(* Logix 5000 project; controller cal1632 1756-L62 rev 16.20; software revision 16.05; part 38 of 57 *)
(* tags used below, declared in another part *)
   FAULT : BOOL;
   p01_param_oven_timer_presets : DINT[32];
   p01_recipe_active : recipe;
   p01r09 : routine;
   p01r09_pb_global_reset : BOOL;
   p02_dint_from_hmi : hmi_dint;
   p02_real_from_hmi : hmi_real;
   p23_ao_servo_ds_jog_vel_cmd : REAL;
   p23_ao_servo_ds_position_cmd : REAL;
   p23_ao_servo_ds_velocity_cmd : REAL;
   p23_ao_servo_ds_zero_offset : REAL;
   p23_ao_servo_os_jog_vel_cmd : REAL;
   p23_ao_servo_os_position_cmd : REAL;
   p23_ao_servo_os_velocity_cmd : REAL;
   p23_ao_servo_os_zero_offset : REAL;
   p23_di_servo_ds : servo_di;
   p23_di_servo_os : servo_di;
   p23_di_vfd_jog_fwd : BOOL;
   p23_di_vfd_jog_rev : BOOL;
   p23_do_servo_ds : servo_do;
   p23_do_servo_os : servo_do;
   p23_param_lfl_hhl : REAL;
   p23_param_lfl_hl : REAL;
   p23_param_zone_pressure : REAL;
   p23r09 : routine;
   p23r09_mode_run : BOOL;
   p23r09_timer_fault : TIMER[4];
   p23r09_web_wet_ctrl_toggle : SYS_Toggle;
   p23r10 : routine;
   p23r10_timer_fault : TIMER[4];
   p23r10_timer_warning : TIMER[4];
   p23r11 : routine;
   p23r11_impreg_gap_os : REAL;
   p23r11_offsets : REAL[100];
   p23r11_permissive_jog : BOOL;
   p23r11_pos_offset : REAL;
   p23r11_request_jog_fwd : BOOL;
   p23r11_request_jog_rev : BOOL;
   p23r11_request_position : BOOL;
   p23r11_request_start : BOOL;
   p23r11_request_zero : BOOL;
   p23r11_selected_position : REAL;
   p23r11_servo_not_ready : BOOL;
   p23r11_servo_status_ab : BOOL;
   p23r11_servo_status_af : BOOL;
   p23r11_servo_status_bb : BOOL;
   p23r11_timer : TIMER[4];
   p23r11_timer_fault : TIMER[4];
   p23r11_timer_warning : TIMER[4];
   p23r12 : routine;
   p23r12_impreg_gap_ds : REAL;
   p23r12_offsets : REAL[100];
   p23r12_permissive_jog : BOOL;
   p23r12_pos_offset : REAL;
   p23r12_request_jog_fwd : BOOL;
   p23r12_request_jog_rev : BOOL;
   p23r12_request_position : BOOL;
   p23r12_request_start : BOOL;
   p23r12_request_zero : BOOL;
   p23r12_selected_position : REAL;
   p23r12_servo_not_ready : BOOL;
   p23r12_servo_status_ab : BOOL;
   p23r12_servo_status_af : BOOL;
   p23r12_servo_status_bb : BOOL;
   p23r12_timer : TIMER[4];
   p23r12_timer_fault : TIMER[4];
   p23r12_timer_warning : TIMER[4];
   p23r15_pid_tension_control : BOOL;
(* P23_Impreg, continued *)

ROUTINE R09_Modes   (* ladder *)
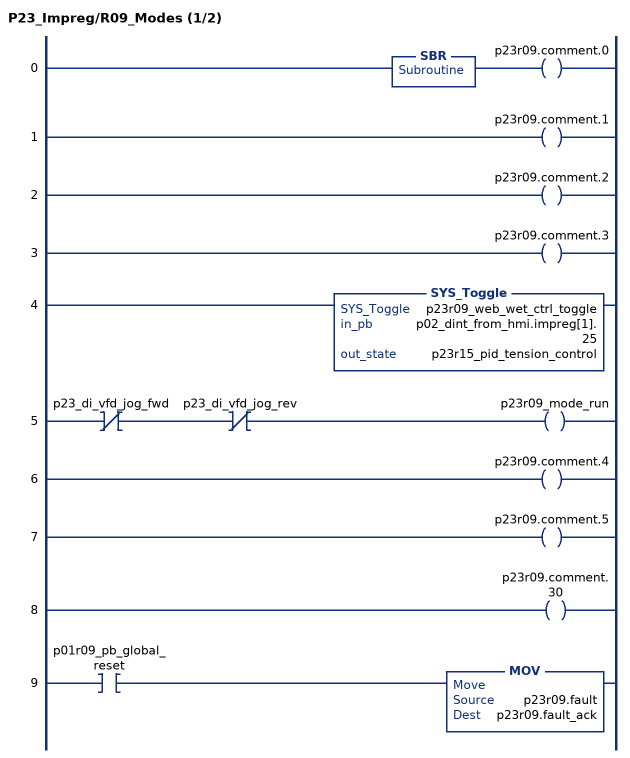
   0: SBR()OTE(p23r09.comment.0);
   1: OTE(p23r09.comment.1);
   2: OTE(p23r09.comment.2);
   3: OTE(p23r09.comment.3);
   4: SYS_Toggle(p23r09_web_wet_ctrl_toggle,p02_dint_from_hmi.impreg[1].25,p23r15_pid_tension_control);
   5: XIO(p23_di_vfd_jog_fwd)XIO(p23_di_vfd_jog_rev)OTE(p23r09_mode_run);
   6: OTE(p23r09.comment.4);
   7: OTE(p23r09.comment.5);
   8: OTE(p23r09.comment.30);
   9: XIC(p01r09_pb_global_reset)MOV(p23r09.fault,p23r09.fault_ack);
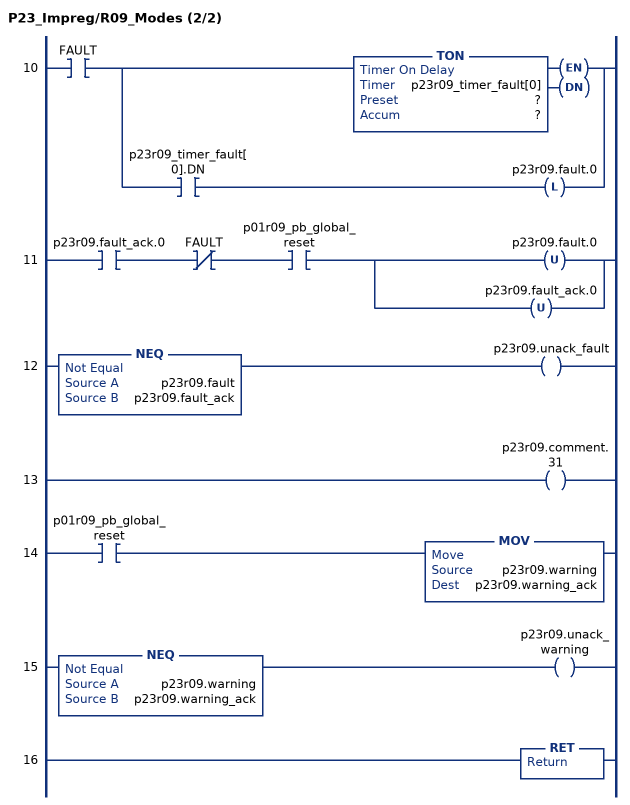
   10: XIC(FAULT)[TON(p23r09_timer_fault[0],?,?) ,XIC(p23r09_timer_fault[0].DN) OTL(p23r09.fault.0) ];
   11: XIC(p23r09.fault_ack.0)XIO(FAULT)XIC(p01r09_pb_global_reset)[OTU(p23r09.fault.0) ,OTU(p23r09.fault_ack.0) ];
   12: NEQ(p23r09.fault,p23r09.fault_ack)OTE(p23r09.unack_fault);
   13: OTE(p23r09.comment.31);
   14: XIC(p01r09_pb_global_reset)MOV(p23r09.warning,p23r09.warning_ack);
   15: NEQ(p23r09.warning,p23r09.warning_ack)OTE(p23r09.unack_warning);
   16: RET();
END_ROUTINE

ROUTINE R10_Parameters   (* ladder *)
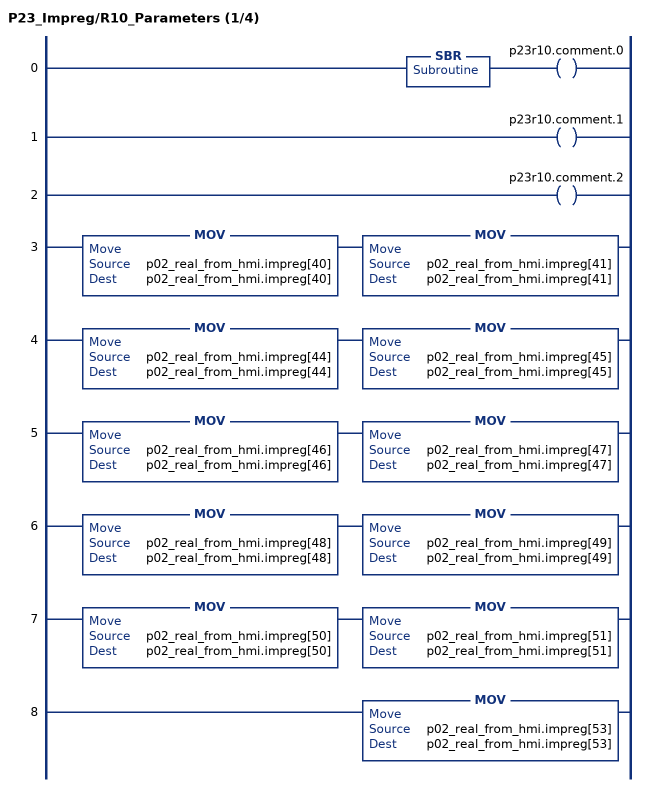
   0: SBR()OTE(p23r10.comment.0);
   1: OTE(p23r10.comment.1);
   2: OTE(p23r10.comment.2);
   3: MOV(p02_real_from_hmi.impreg[40],p02_real_from_hmi.impreg[40])MOV(p02_real_from_hmi.impreg[41],p02_real_from_hmi.impreg[41]);
   4: MOV(p02_real_from_hmi.impreg[44],p02_real_from_hmi.impreg[44])MOV(p02_real_from_hmi.impreg[45],p02_real_from_hmi.impreg[45]);
   5: MOV(p02_real_from_hmi.impreg[46],p02_real_from_hmi.impreg[46])MOV(p02_real_from_hmi.impreg[47],p02_real_from_hmi.impreg[47]);
   6: MOV(p02_real_from_hmi.impreg[48],p02_real_from_hmi.impreg[48])MOV(p02_real_from_hmi.impreg[49],p02_real_from_hmi.impreg[49]);
   7: MOV(p02_real_from_hmi.impreg[50],p02_real_from_hmi.impreg[50])MOV(p02_real_from_hmi.impreg[51],p02_real_from_hmi.impreg[51]);
   8: MOV(p02_real_from_hmi.impreg[53],p02_real_from_hmi.impreg[53]);
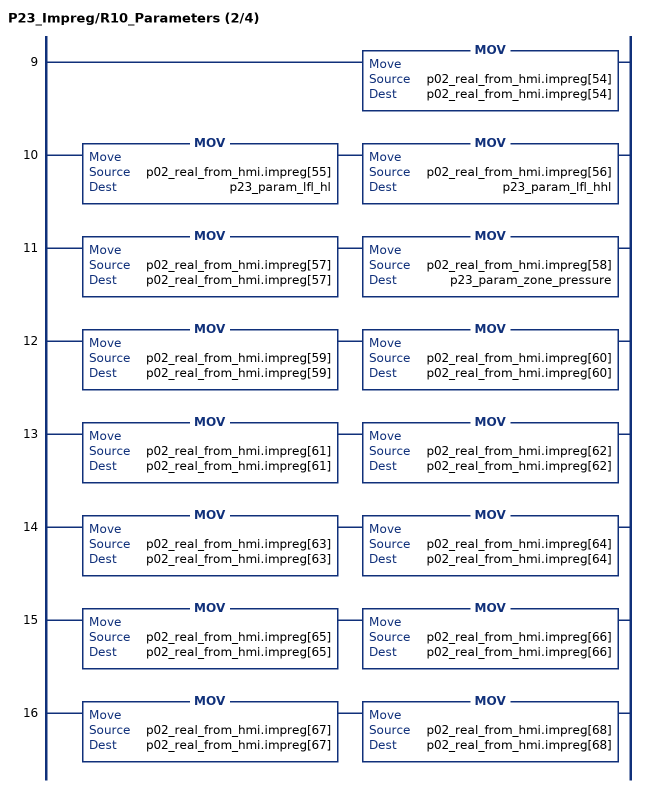
   9: MOV(p02_real_from_hmi.impreg[54],p02_real_from_hmi.impreg[54]);
   10: MOV(p02_real_from_hmi.impreg[55],p23_param_lfl_hl)MOV(p02_real_from_hmi.impreg[56],p23_param_lfl_hhl);
   11: MOV(p02_real_from_hmi.impreg[57],p02_real_from_hmi.impreg[57])MOV(p02_real_from_hmi.impreg[58],p23_param_zone_pressure);
   12: MOV(p02_real_from_hmi.impreg[59],p02_real_from_hmi.impreg[59])MOV(p02_real_from_hmi.impreg[60],p02_real_from_hmi.impreg[60]);
   13: MOV(p02_real_from_hmi.impreg[61],p02_real_from_hmi.impreg[61])MOV(p02_real_from_hmi.impreg[62],p02_real_from_hmi.impreg[62]);
   14: MOV(p02_real_from_hmi.impreg[63],p02_real_from_hmi.impreg[63])MOV(p02_real_from_hmi.impreg[64],p02_real_from_hmi.impreg[64]);
   15: MOV(p02_real_from_hmi.impreg[65],p02_real_from_hmi.impreg[65])MOV(p02_real_from_hmi.impreg[66],p02_real_from_hmi.impreg[66]);
   16: MOV(p02_real_from_hmi.impreg[67],p02_real_from_hmi.impreg[67])MOV(p02_real_from_hmi.impreg[68],p02_real_from_hmi.impreg[68]);
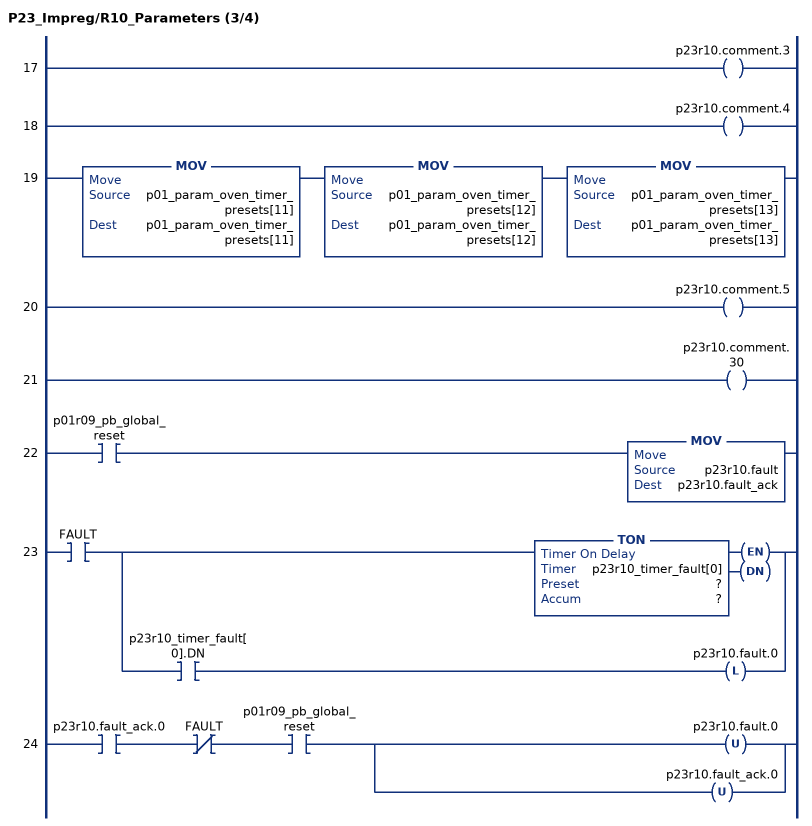
   17: OTE(p23r10.comment.3);
   18: OTE(p23r10.comment.4);
   19: MOV(p01_param_oven_timer_presets[11],p01_param_oven_timer_presets[11])MOV(p01_param_oven_timer_presets[12],p01_param_oven_timer_presets[12])MOV(p01_param_oven_timer_presets[13],p01_param_oven_timer_presets[13]);
   20: OTE(p23r10.comment.5);
   21: OTE(p23r10.comment.30);
   22: XIC(p01r09_pb_global_reset)MOV(p23r10.fault,p23r10.fault_ack);
   23: XIC(FAULT)[TON(p23r10_timer_fault[0],?,?) ,XIC(p23r10_timer_fault[0].DN) OTL(p23r10.fault.0) ];
   24: XIC(p23r10.fault_ack.0)XIO(FAULT)XIC(p01r09_pb_global_reset)[OTU(p23r10.fault.0) ,OTU(p23r10.fault_ack.0) ];
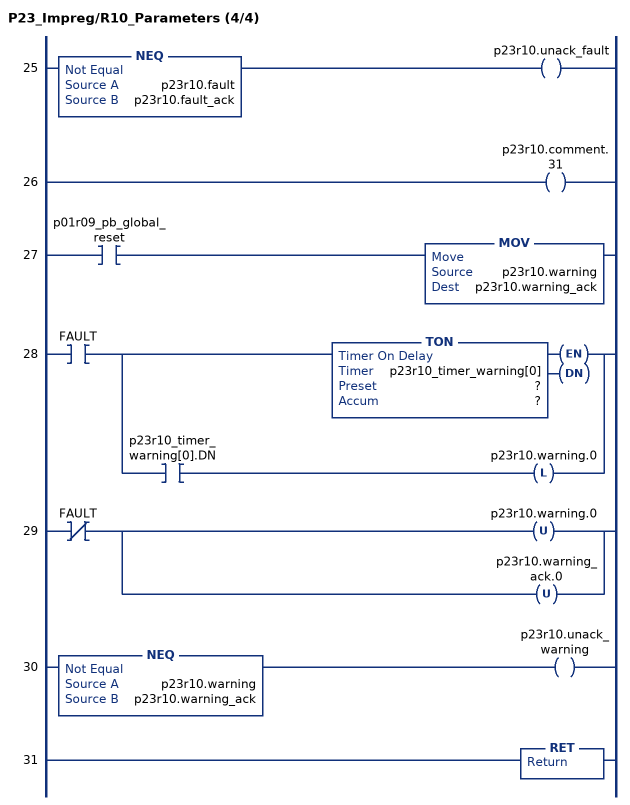
   25: NEQ(p23r10.fault,p23r10.fault_ack)OTE(p23r10.unack_fault);
   26: OTE(p23r10.comment.31);
   27: XIC(p01r09_pb_global_reset)MOV(p23r10.warning,p23r10.warning_ack);
   28: XIC(FAULT)[TON(p23r10_timer_warning[0],?,?) ,XIC(p23r10_timer_warning[0].DN) OTL(p23r10.warning.0) ];
   29: XIO(FAULT)[OTU(p23r10.warning.0) ,OTU(p23r10.warning_ack.0) ];
   30: NEQ(p23r10.warning,p23r10.warning_ack)OTE(p23r10.unack_warning);
   31: RET();
END_ROUTINE

ROUTINE R11_Servo_Operator_Side   (* ladder *)
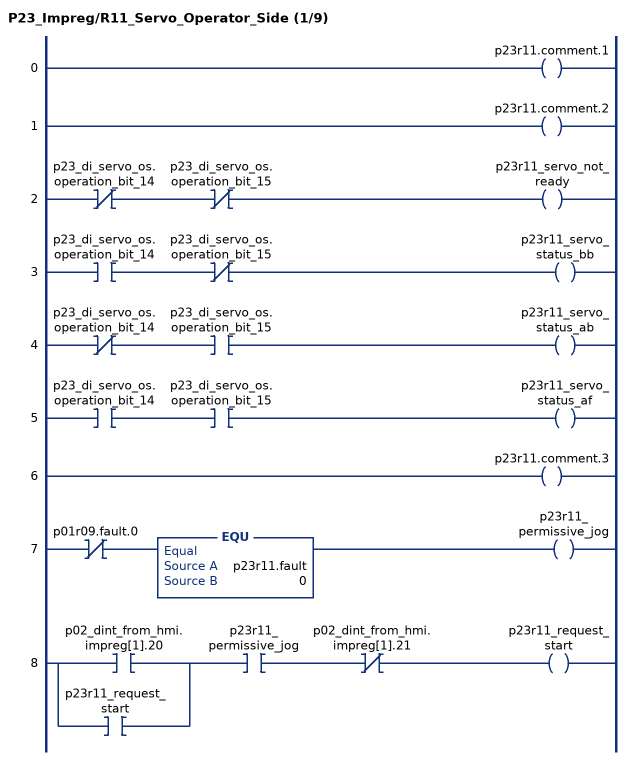
   0: OTE(p23r11.comment.1);
   1: OTE(p23r11.comment.2);
   2: XIO(p23_di_servo_os.operation_bit_14)XIO(p23_di_servo_os.operation_bit_15)OTE(p23r11_servo_not_ready);
   3: XIC(p23_di_servo_os.operation_bit_14)XIO(p23_di_servo_os.operation_bit_15)OTE(p23r11_servo_status_bb);
   4: XIO(p23_di_servo_os.operation_bit_14)XIC(p23_di_servo_os.operation_bit_15)OTE(p23r11_servo_status_ab);
   5: XIC(p23_di_servo_os.operation_bit_14)XIC(p23_di_servo_os.operation_bit_15)OTE(p23r11_servo_status_af);
   6: OTE(p23r11.comment.3);
   7: XIO(p01r09.fault.0)EQU(p23r11.fault,0)OTE(p23r11_permissive_jog);
   8: [XIC(p02_dint_from_hmi.impreg[1].20) ,XIC(p23r11_request_start) ]XIC(p23r11_permissive_jog)XIO(p02_dint_from_hmi.impreg[1].21)OTE(p23r11_request_start);
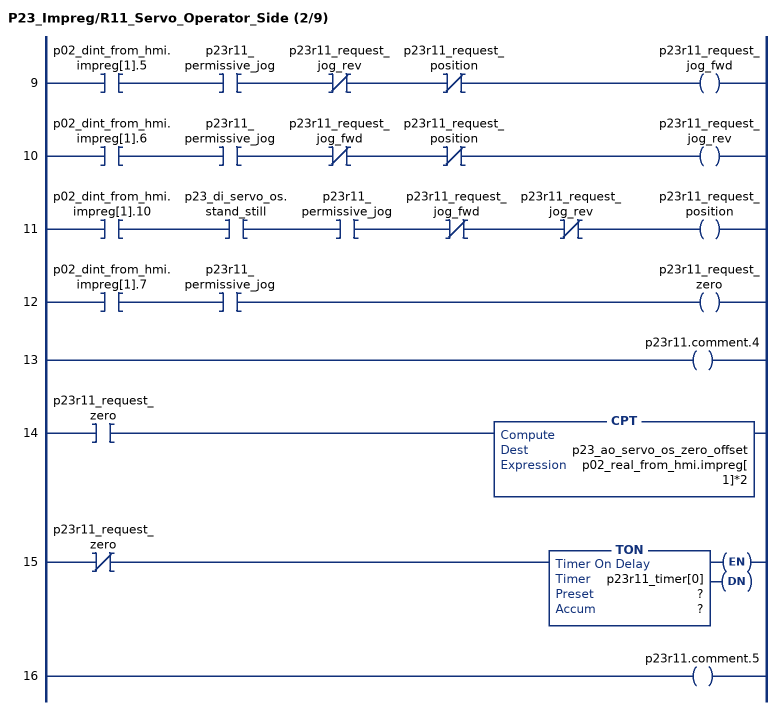
   9: XIC(p02_dint_from_hmi.impreg[1].5)XIC(p23r11_permissive_jog)XIO(p23r11_request_jog_rev)XIO(p23r11_request_position)OTE(p23r11_request_jog_fwd);
   10: XIC(p02_dint_from_hmi.impreg[1].6)XIC(p23r11_permissive_jog)XIO(p23r11_request_jog_fwd)XIO(p23r11_request_position)OTE(p23r11_request_jog_rev);
   11: XIC(p02_dint_from_hmi.impreg[1].10)XIC(p23_di_servo_os.stand_still)XIC(p23r11_permissive_jog)XIO(p23r11_request_jog_fwd)XIO(p23r11_request_jog_rev)OTE(p23r11_request_position);
   12: XIC(p02_dint_from_hmi.impreg[1].7)XIC(p23r11_permissive_jog)OTE(p23r11_request_zero);
   13: OTE(p23r11.comment.4);
   14: XIC(p23r11_request_zero)CPT(p23_ao_servo_os_zero_offset,p02_real_from_hmi.impreg[1]*2);
   15: XIO(p23r11_request_zero)TON(p23r11_timer[0],?,?);
   16: OTE(p23r11.comment.5);
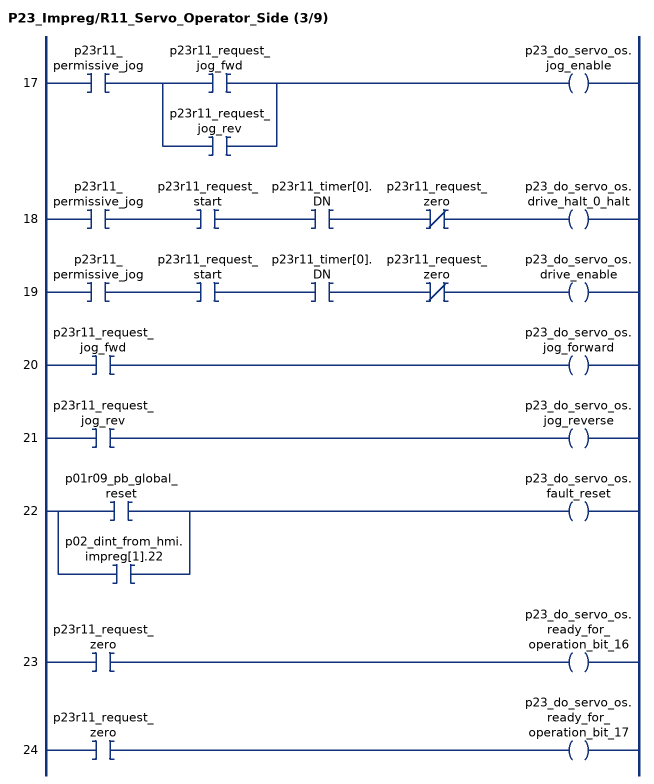
   17: XIC(p23r11_permissive_jog)[XIC(p23r11_request_jog_fwd) ,XIC(p23r11_request_jog_rev) ]OTE(p23_do_servo_os.jog_enable);
   18: XIC(p23r11_permissive_jog)XIC(p23r11_request_start)XIC(p23r11_timer[0].DN)XIO(p23r11_request_zero)OTE(p23_do_servo_os.drive_halt_0_halt);
   19: XIC(p23r11_permissive_jog)XIC(p23r11_request_start)XIC(p23r11_timer[0].DN)XIO(p23r11_request_zero)OTE(p23_do_servo_os.drive_enable);
   20: XIC(p23r11_request_jog_fwd)OTE(p23_do_servo_os.jog_forward);
   21: XIC(p23r11_request_jog_rev)OTE(p23_do_servo_os.jog_reverse);
   22: [XIC(p01r09_pb_global_reset) ,XIC(p02_dint_from_hmi.impreg[1].22) ]OTE(p23_do_servo_os.fault_reset);
   23: XIC(p23r11_request_zero)OTE(p23_do_servo_os.ready_for_operation_bit_16);
   24: XIC(p23r11_request_zero)OTE(p23_do_servo_os.ready_for_operation_bit_17);
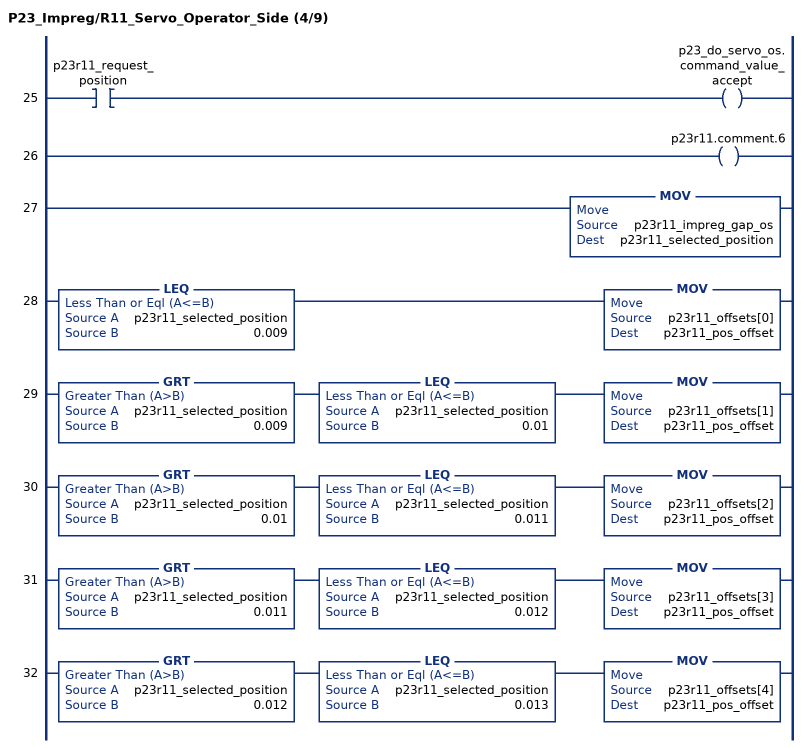
   25: XIC(p23r11_request_position)OTE(p23_do_servo_os.command_value_accept);
   26: OTE(p23r11.comment.6);
   27: MOV(p23r11_impreg_gap_os,p23r11_selected_position);
   28: LEQ(p23r11_selected_position,0.009)MOV(p23r11_offsets[0],p23r11_pos_offset);
   29: GRT(p23r11_selected_position,0.009)LEQ(p23r11_selected_position,0.01)MOV(p23r11_offsets[1],p23r11_pos_offset);
   30: GRT(p23r11_selected_position,0.01)LEQ(p23r11_selected_position,0.011)MOV(p23r11_offsets[2],p23r11_pos_offset);
   31: GRT(p23r11_selected_position,0.011)LEQ(p23r11_selected_position,0.012)MOV(p23r11_offsets[3],p23r11_pos_offset);
   32: GRT(p23r11_selected_position,0.012)LEQ(p23r11_selected_position,0.013)MOV(p23r11_offsets[4],p23r11_pos_offset);
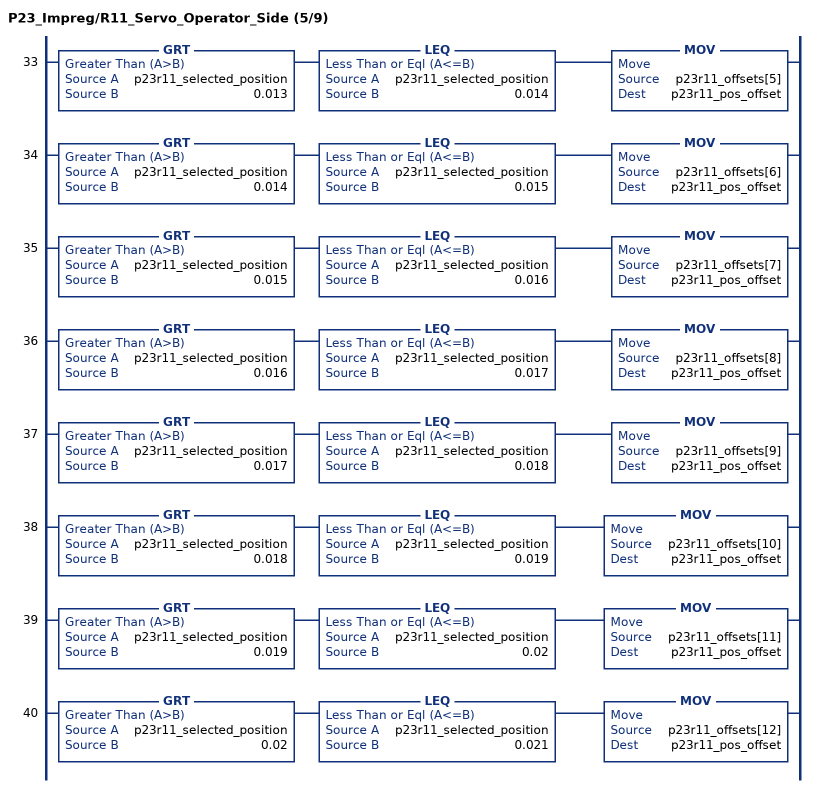
   33: GRT(p23r11_selected_position,0.013)LEQ(p23r11_selected_position,0.014)MOV(p23r11_offsets[5],p23r11_pos_offset);
   34: GRT(p23r11_selected_position,0.014)LEQ(p23r11_selected_position,0.015)MOV(p23r11_offsets[6],p23r11_pos_offset);
   35: GRT(p23r11_selected_position,0.015)LEQ(p23r11_selected_position,0.016)MOV(p23r11_offsets[7],p23r11_pos_offset);
   36: GRT(p23r11_selected_position,0.016)LEQ(p23r11_selected_position,0.017)MOV(p23r11_offsets[8],p23r11_pos_offset);
   37: GRT(p23r11_selected_position,0.017)LEQ(p23r11_selected_position,0.018)MOV(p23r11_offsets[9],p23r11_pos_offset);
   38: GRT(p23r11_selected_position,0.018)LEQ(p23r11_selected_position,0.019)MOV(p23r11_offsets[10],p23r11_pos_offset);
   39: GRT(p23r11_selected_position,0.019)LEQ(p23r11_selected_position,0.02)MOV(p23r11_offsets[11],p23r11_pos_offset);
   40: GRT(p23r11_selected_position,0.02)LEQ(p23r11_selected_position,0.021)MOV(p23r11_offsets[12],p23r11_pos_offset);
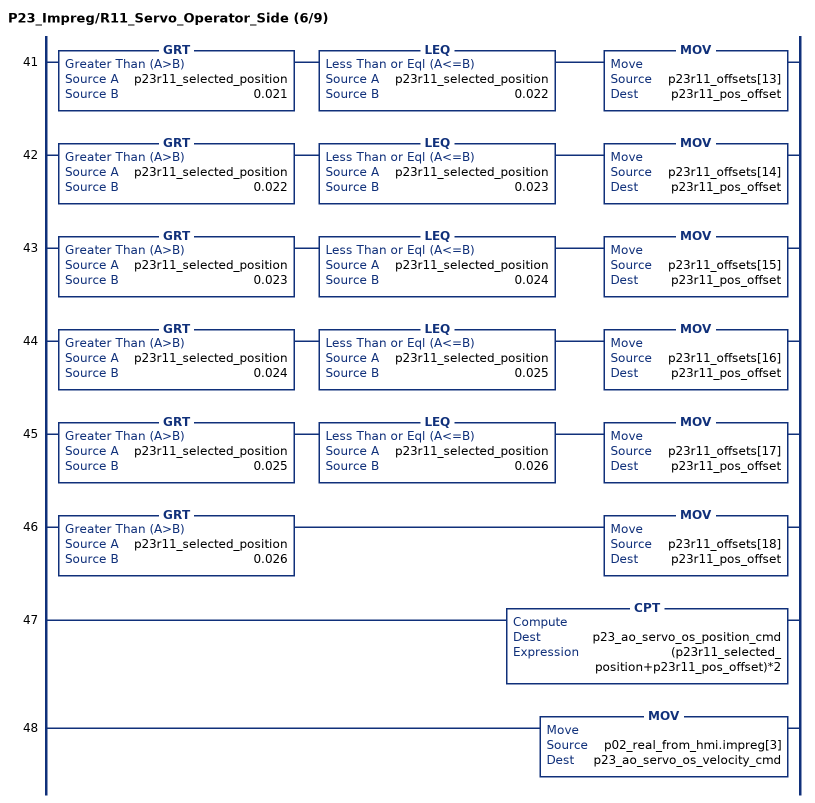
   41: GRT(p23r11_selected_position,0.021)LEQ(p23r11_selected_position,0.022)MOV(p23r11_offsets[13],p23r11_pos_offset);
   42: GRT(p23r11_selected_position,0.022)LEQ(p23r11_selected_position,0.023)MOV(p23r11_offsets[14],p23r11_pos_offset);
   43: GRT(p23r11_selected_position,0.023)LEQ(p23r11_selected_position,0.024)MOV(p23r11_offsets[15],p23r11_pos_offset);
   44: GRT(p23r11_selected_position,0.024)LEQ(p23r11_selected_position,0.025)MOV(p23r11_offsets[16],p23r11_pos_offset);
   45: GRT(p23r11_selected_position,0.025)LEQ(p23r11_selected_position,0.026)MOV(p23r11_offsets[17],p23r11_pos_offset);
   46: GRT(p23r11_selected_position,0.026)MOV(p23r11_offsets[18],p23r11_pos_offset);
   47: CPT(p23_ao_servo_os_position_cmd,(p23r11_selected_position+p23r11_pos_offset)*2);
   48: MOV(p02_real_from_hmi.impreg[3],p23_ao_servo_os_velocity_cmd);
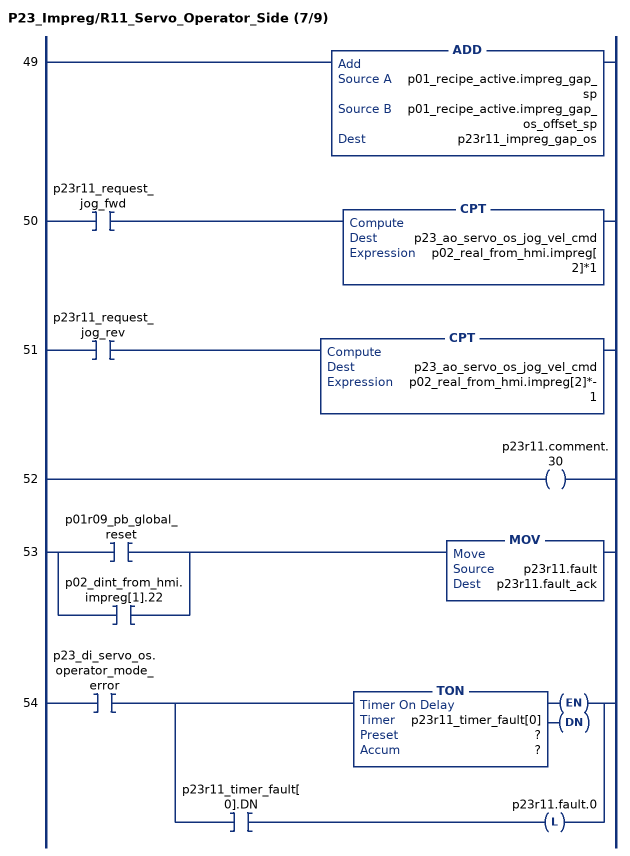
   49: ADD(p01_recipe_active.impreg_gap_sp,p01_recipe_active.impreg_gap_os_offset_sp,p23r11_impreg_gap_os);
   50: XIC(p23r11_request_jog_fwd)CPT(p23_ao_servo_os_jog_vel_cmd,p02_real_from_hmi.impreg[2]*1);
   51: XIC(p23r11_request_jog_rev)CPT(p23_ao_servo_os_jog_vel_cmd,p02_real_from_hmi.impreg[2]*-1);
   52: OTE(p23r11.comment.30);
   53: [XIC(p01r09_pb_global_reset) ,XIC(p02_dint_from_hmi.impreg[1].22) ]MOV(p23r11.fault,p23r11.fault_ack);
   54: XIC(p23_di_servo_os.operator_mode_error)[TON(p23r11_timer_fault[0],?,?) ,XIC(p23r11_timer_fault[0].DN) OTL(p23r11.fault.0) ];
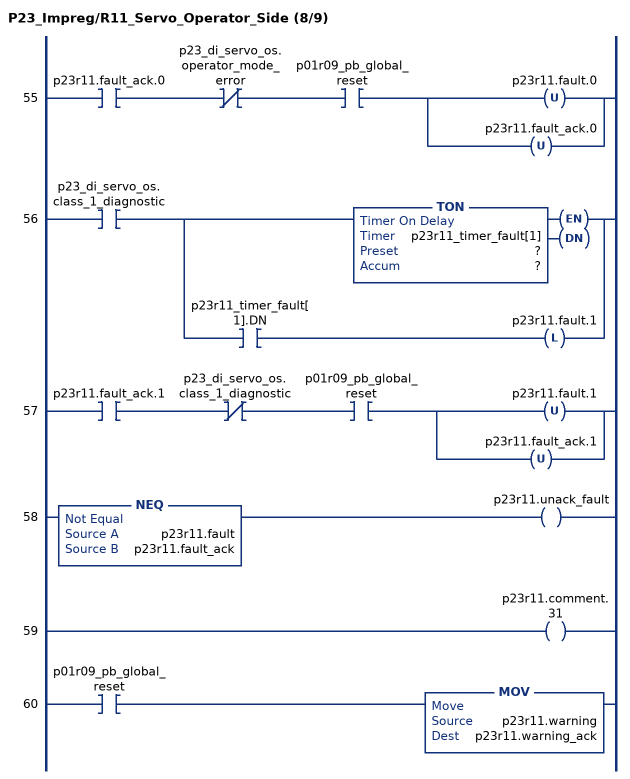
   55: XIC(p23r11.fault_ack.0)XIO(p23_di_servo_os.operator_mode_error)XIC(p01r09_pb_global_reset)[OTU(p23r11.fault.0) ,OTU(p23r11.fault_ack.0) ];
   56: XIC(p23_di_servo_os.class_1_diagnostic)[TON(p23r11_timer_fault[1],?,?) ,XIC(p23r11_timer_fault[1].DN) OTL(p23r11.fault.1) ];
   57: XIC(p23r11.fault_ack.1)XIO(p23_di_servo_os.class_1_diagnostic)XIC(p01r09_pb_global_reset)[OTU(p23r11.fault.1) ,OTU(p23r11.fault_ack.1) ];
   58: NEQ(p23r11.fault,p23r11.fault_ack)OTE(p23r11.unack_fault);
   59: OTE(p23r11.comment.31);
   60: XIC(p01r09_pb_global_reset)MOV(p23r11.warning,p23r11.warning_ack);
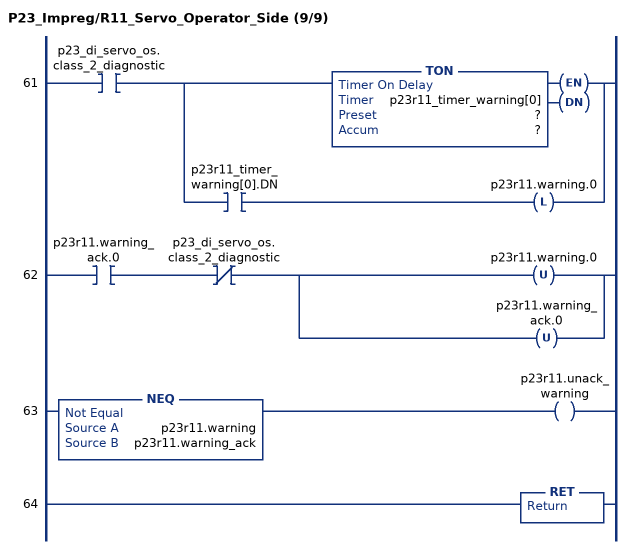
   61: XIC(p23_di_servo_os.class_2_diagnostic)[TON(p23r11_timer_warning[0],?,?) ,XIC(p23r11_timer_warning[0].DN) OTL(p23r11.warning.0) ];
   62: XIC(p23r11.warning_ack.0)XIO(p23_di_servo_os.class_2_diagnostic)[OTU(p23r11.warning.0) ,OTU(p23r11.warning_ack.0) ];
   63: NEQ(p23r11.warning,p23r11.warning_ack)OTE(p23r11.unack_warning);
   64: RET();
END_ROUTINE

ROUTINE R12_Servo_Drive_Side   (* ladder *)
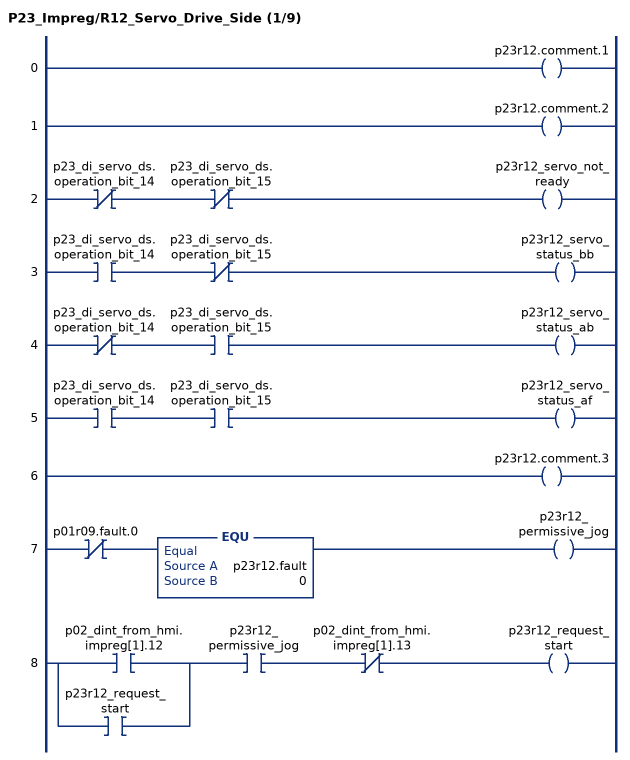
   0: OTE(p23r12.comment.1);
   1: OTE(p23r12.comment.2);
   2: XIO(p23_di_servo_ds.operation_bit_14)XIO(p23_di_servo_ds.operation_bit_15)OTE(p23r12_servo_not_ready);
   3: XIC(p23_di_servo_ds.operation_bit_14)XIO(p23_di_servo_ds.operation_bit_15)OTE(p23r12_servo_status_bb);
   4: XIO(p23_di_servo_ds.operation_bit_14)XIC(p23_di_servo_ds.operation_bit_15)OTE(p23r12_servo_status_ab);
   5: XIC(p23_di_servo_ds.operation_bit_14)XIC(p23_di_servo_ds.operation_bit_15)OTE(p23r12_servo_status_af);
   6: OTE(p23r12.comment.3);
   7: XIO(p01r09.fault.0)EQU(p23r12.fault,0)OTE(p23r12_permissive_jog);
   8: [XIC(p02_dint_from_hmi.impreg[1].12) ,XIC(p23r12_request_start) ]XIC(p23r12_permissive_jog)XIO(p02_dint_from_hmi.impreg[1].13)OTE(p23r12_request_start);
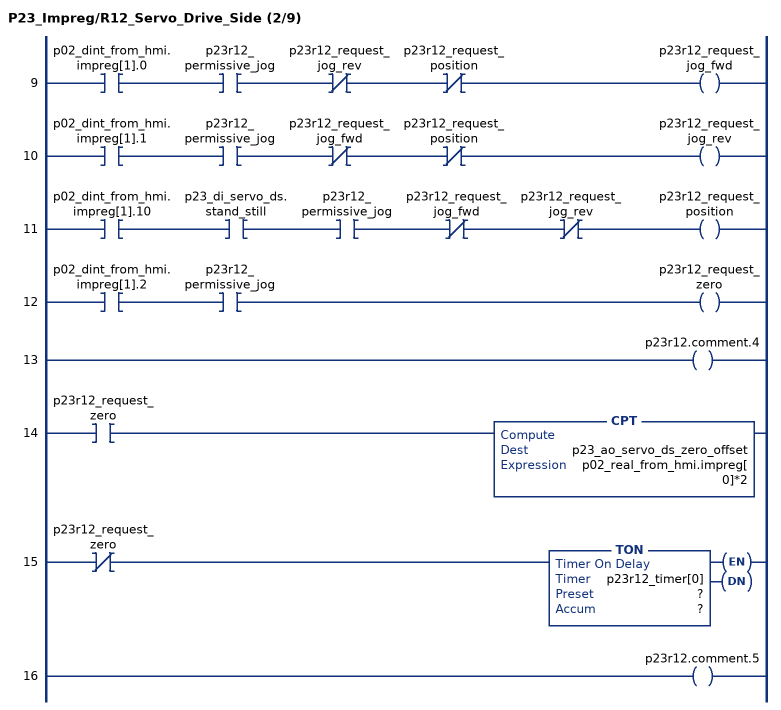
   9: XIC(p02_dint_from_hmi.impreg[1].0)XIC(p23r12_permissive_jog)XIO(p23r12_request_jog_rev)XIO(p23r12_request_position)OTE(p23r12_request_jog_fwd);
   10: XIC(p02_dint_from_hmi.impreg[1].1)XIC(p23r12_permissive_jog)XIO(p23r12_request_jog_fwd)XIO(p23r12_request_position)OTE(p23r12_request_jog_rev);
   11: XIC(p02_dint_from_hmi.impreg[1].10)XIC(p23_di_servo_ds.stand_still)XIC(p23r12_permissive_jog)XIO(p23r12_request_jog_fwd)XIO(p23r12_request_jog_rev)OTE(p23r12_request_position);
   12: XIC(p02_dint_from_hmi.impreg[1].2)XIC(p23r12_permissive_jog)OTE(p23r12_request_zero);
   13: OTE(p23r12.comment.4);
   14: XIC(p23r12_request_zero)CPT(p23_ao_servo_ds_zero_offset,p02_real_from_hmi.impreg[0]*2);
   15: XIO(p23r12_request_zero)TON(p23r12_timer[0],?,?);
   16: OTE(p23r12.comment.5);
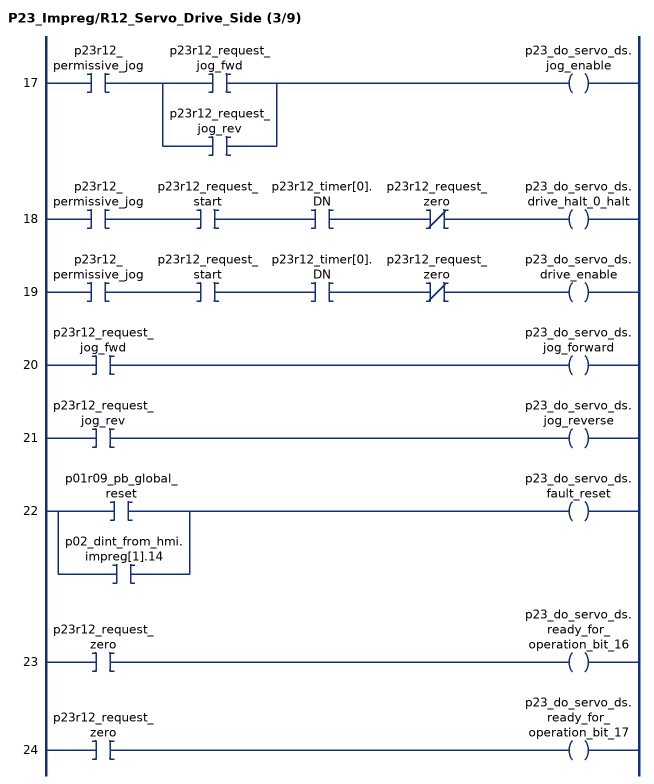
   17: XIC(p23r12_permissive_jog)[XIC(p23r12_request_jog_fwd) ,XIC(p23r12_request_jog_rev) ]OTE(p23_do_servo_ds.jog_enable);
   18: XIC(p23r12_permissive_jog)XIC(p23r12_request_start)XIC(p23r12_timer[0].DN)XIO(p23r12_request_zero)OTE(p23_do_servo_ds.drive_halt_0_halt);
   19: XIC(p23r12_permissive_jog)XIC(p23r12_request_start)XIC(p23r12_timer[0].DN)XIO(p23r12_request_zero)OTE(p23_do_servo_ds.drive_enable);
   20: XIC(p23r12_request_jog_fwd)OTE(p23_do_servo_ds.jog_forward);
   21: XIC(p23r12_request_jog_rev)OTE(p23_do_servo_ds.jog_reverse);
   22: [XIC(p01r09_pb_global_reset) ,XIC(p02_dint_from_hmi.impreg[1].14) ]OTE(p23_do_servo_ds.fault_reset);
   23: XIC(p23r12_request_zero)OTE(p23_do_servo_ds.ready_for_operation_bit_16);
   24: XIC(p23r12_request_zero)OTE(p23_do_servo_ds.ready_for_operation_bit_17);
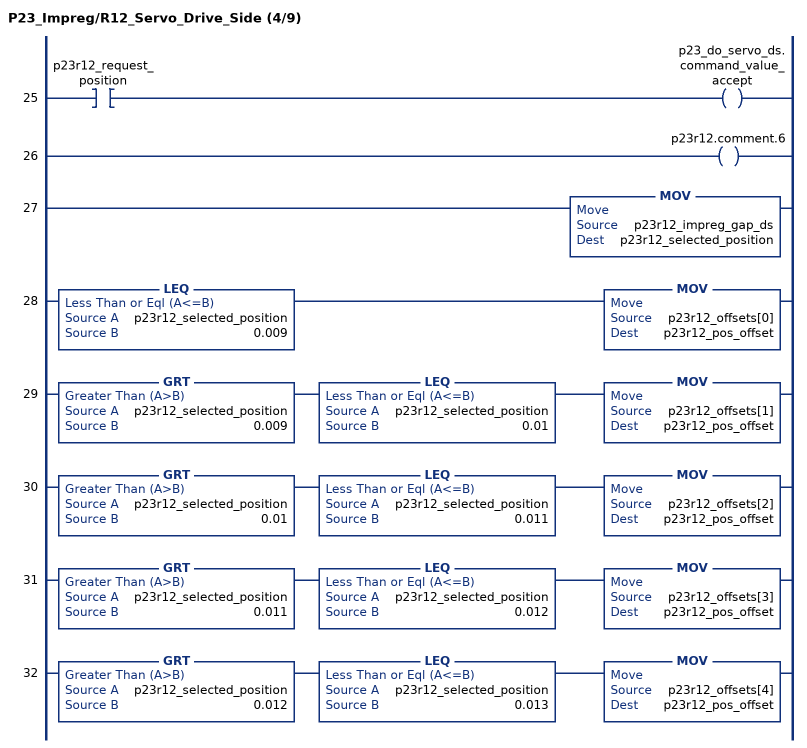
   25: XIC(p23r12_request_position)OTE(p23_do_servo_ds.command_value_accept);
   26: OTE(p23r12.comment.6);
   27: MOV(p23r12_impreg_gap_ds,p23r12_selected_position);
   28: LEQ(p23r12_selected_position,0.009)MOV(p23r12_offsets[0],p23r12_pos_offset);
   29: GRT(p23r12_selected_position,0.009)LEQ(p23r12_selected_position,0.01)MOV(p23r12_offsets[1],p23r12_pos_offset);
   30: GRT(p23r12_selected_position,0.01)LEQ(p23r12_selected_position,0.011)MOV(p23r12_offsets[2],p23r12_pos_offset);
   31: GRT(p23r12_selected_position,0.011)LEQ(p23r12_selected_position,0.012)MOV(p23r12_offsets[3],p23r12_pos_offset);
   32: GRT(p23r12_selected_position,0.012)LEQ(p23r12_selected_position,0.013)MOV(p23r12_offsets[4],p23r12_pos_offset);
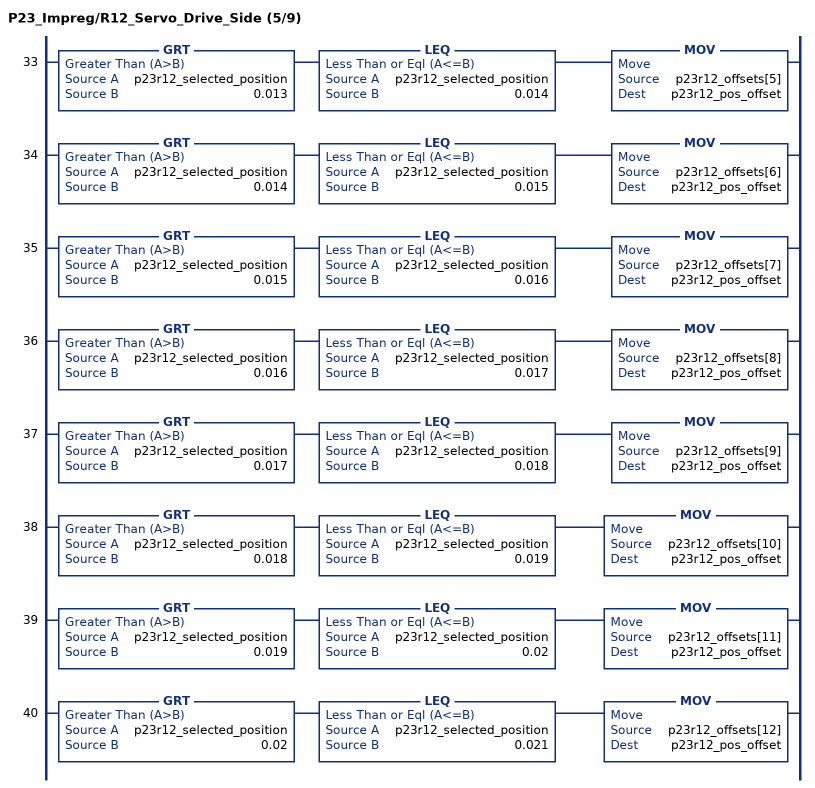
   33: GRT(p23r12_selected_position,0.013)LEQ(p23r12_selected_position,0.014)MOV(p23r12_offsets[5],p23r12_pos_offset);
   34: GRT(p23r12_selected_position,0.014)LEQ(p23r12_selected_position,0.015)MOV(p23r12_offsets[6],p23r12_pos_offset);
   35: GRT(p23r12_selected_position,0.015)LEQ(p23r12_selected_position,0.016)MOV(p23r12_offsets[7],p23r12_pos_offset);
   36: GRT(p23r12_selected_position,0.016)LEQ(p23r12_selected_position,0.017)MOV(p23r12_offsets[8],p23r12_pos_offset);
   37: GRT(p23r12_selected_position,0.017)LEQ(p23r12_selected_position,0.018)MOV(p23r12_offsets[9],p23r12_pos_offset);
   38: GRT(p23r12_selected_position,0.018)LEQ(p23r12_selected_position,0.019)MOV(p23r12_offsets[10],p23r12_pos_offset);
   39: GRT(p23r12_selected_position,0.019)LEQ(p23r12_selected_position,0.02)MOV(p23r12_offsets[11],p23r12_pos_offset);
   40: GRT(p23r12_selected_position,0.02)LEQ(p23r12_selected_position,0.021)MOV(p23r12_offsets[12],p23r12_pos_offset);
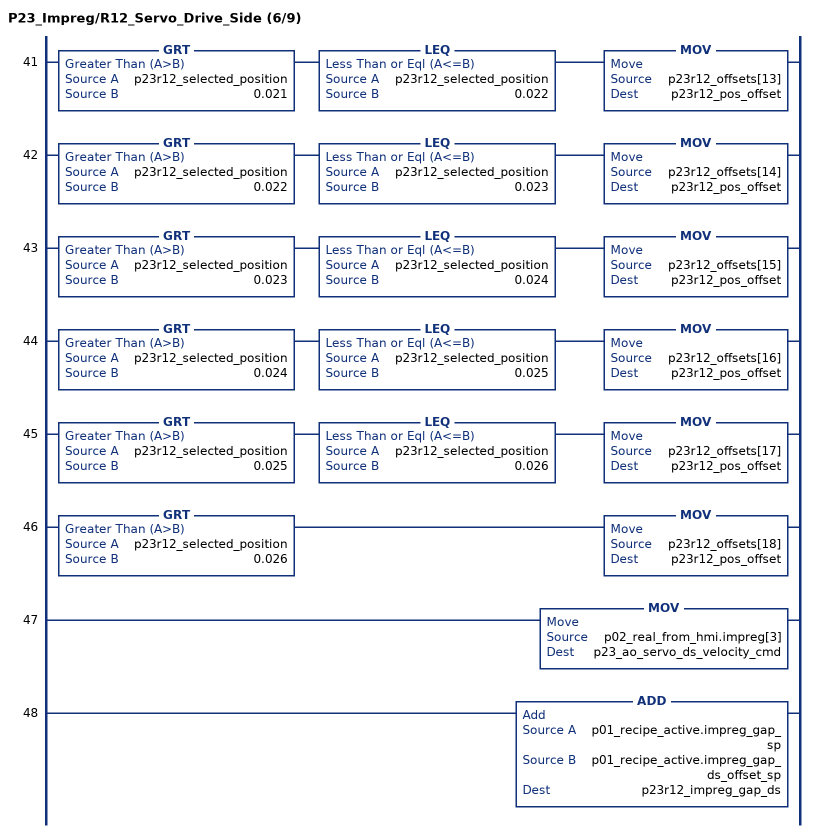
   41: GRT(p23r12_selected_position,0.021)LEQ(p23r12_selected_position,0.022)MOV(p23r12_offsets[13],p23r12_pos_offset);
   42: GRT(p23r12_selected_position,0.022)LEQ(p23r12_selected_position,0.023)MOV(p23r12_offsets[14],p23r12_pos_offset);
   43: GRT(p23r12_selected_position,0.023)LEQ(p23r12_selected_position,0.024)MOV(p23r12_offsets[15],p23r12_pos_offset);
   44: GRT(p23r12_selected_position,0.024)LEQ(p23r12_selected_position,0.025)MOV(p23r12_offsets[16],p23r12_pos_offset);
   45: GRT(p23r12_selected_position,0.025)LEQ(p23r12_selected_position,0.026)MOV(p23r12_offsets[17],p23r12_pos_offset);
   46: GRT(p23r12_selected_position,0.026)MOV(p23r12_offsets[18],p23r12_pos_offset);
   47: MOV(p02_real_from_hmi.impreg[3],p23_ao_servo_ds_velocity_cmd);
   48: ADD(p01_recipe_active.impreg_gap_sp,p01_recipe_active.impreg_gap_ds_offset_sp,p23r12_impreg_gap_ds);
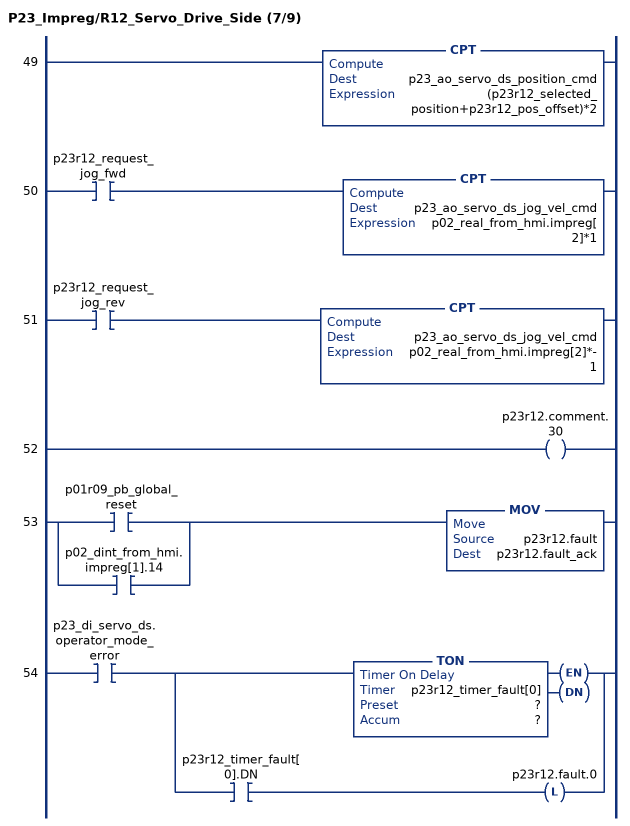
   49: CPT(p23_ao_servo_ds_position_cmd,(p23r12_selected_position+p23r12_pos_offset)*2);
   50: XIC(p23r12_request_jog_fwd)CPT(p23_ao_servo_ds_jog_vel_cmd,p02_real_from_hmi.impreg[2]*1);
   51: XIC(p23r12_request_jog_rev)CPT(p23_ao_servo_ds_jog_vel_cmd,p02_real_from_hmi.impreg[2]*-1);
   52: OTE(p23r12.comment.30);
   53: [XIC(p01r09_pb_global_reset) ,XIC(p02_dint_from_hmi.impreg[1].14) ]MOV(p23r12.fault,p23r12.fault_ack);
   54: XIC(p23_di_servo_ds.operator_mode_error)[TON(p23r12_timer_fault[0],?,?) ,XIC(p23r12_timer_fault[0].DN) OTL(p23r12.fault.0) ];
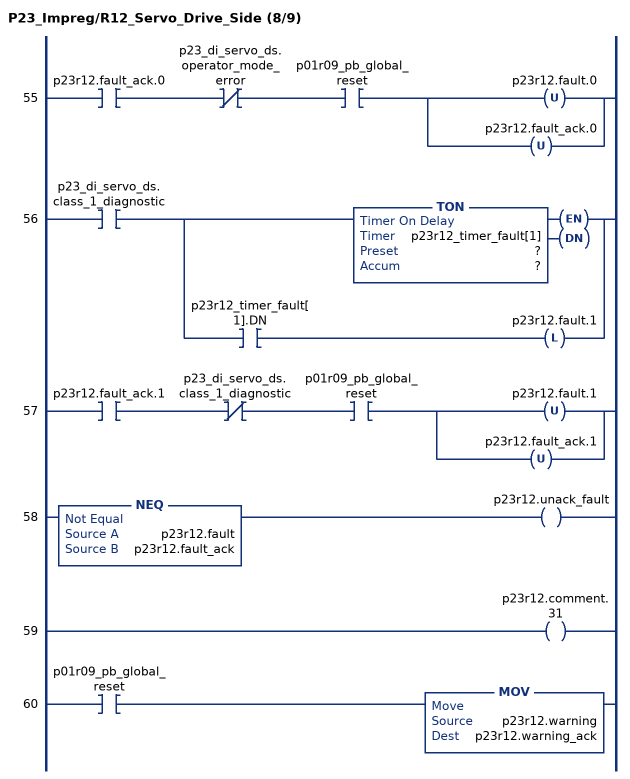
   55: XIC(p23r12.fault_ack.0)XIO(p23_di_servo_ds.operator_mode_error)XIC(p01r09_pb_global_reset)[OTU(p23r12.fault.0) ,OTU(p23r12.fault_ack.0) ];
   56: XIC(p23_di_servo_ds.class_1_diagnostic)[TON(p23r12_timer_fault[1],?,?) ,XIC(p23r12_timer_fault[1].DN) OTL(p23r12.fault.1) ];
   57: XIC(p23r12.fault_ack.1)XIO(p23_di_servo_ds.class_1_diagnostic)XIC(p01r09_pb_global_reset)[OTU(p23r12.fault.1) ,OTU(p23r12.fault_ack.1) ];
   58: NEQ(p23r12.fault,p23r12.fault_ack)OTE(p23r12.unack_fault);
   59: OTE(p23r12.comment.31);
   60: XIC(p01r09_pb_global_reset)MOV(p23r12.warning,p23r12.warning_ack);
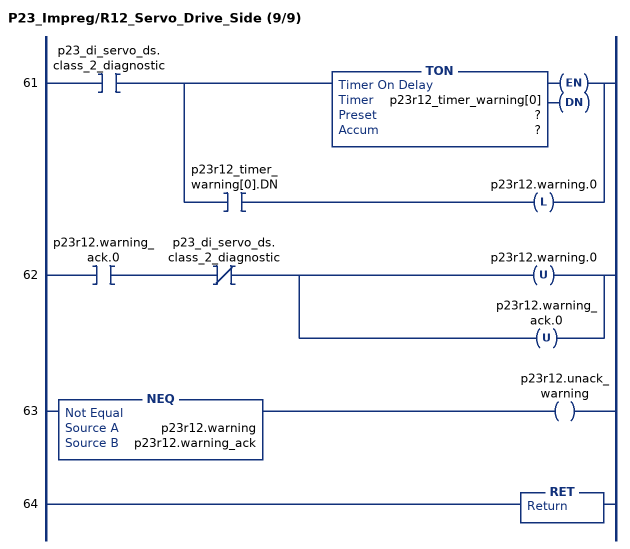
   61: XIC(p23_di_servo_ds.class_2_diagnostic)[TON(p23r12_timer_warning[0],?,?) ,XIC(p23r12_timer_warning[0].DN) OTL(p23r12.warning.0) ];
   62: XIC(p23r12.warning_ack.0)XIO(p23_di_servo_ds.class_2_diagnostic)[OTU(p23r12.warning.0) ,OTU(p23r12.warning_ack.0) ];
   63: NEQ(p23r12.warning,p23r12.warning_ack)OTE(p23r12.unack_warning);
   64: RET();
END_ROUTINE
